(* IEC 61131-3 sources: beeguard/reference, 3 files *)

(* ---- analog_alarm.st ---- *)
FUNCTION_BLOCK BG_ALM_ANA
(*==========================================================================
BG_ALM_ANA - beeguard analog alarm.
Watches one REAL for up to six alarm conditions. Each condition is handled by
its own BG_ALM_DIG instance, so each one has the complete ISA-18.2 behaviour
(acknowledge, latch, shelve, priority, time stamps, count, chatter) and can be
acknowledged or shelved separately. Names follow BG_ALM_DIG (IN_, CFG_, CMD_OP_,
CMD_PG_, STS_, VAL_, TS_).

CONDITIONS (each enabled separately; HH and H may be in alarm at the same time)
	HH      above CFG_HH_SP; normal again below CFG_HH_SP - CFG_DEADBAND
	H       above CFG_H_SP;  normal again below CFG_H_SP  - CFG_DEADBAND
	L       below CFG_L_SP;  normal again above CFG_L_SP  + CFG_DEADBAND
	LL      below CFG_LL_SP; normal again above CFG_LL_SP + CFG_DEADBAND
	ROC_UP  rising faster than CFG_ROC_UP_SP units per second
	ROC_DN  falling faster than CFG_ROC_DN_SP units per second (enter it positive)
	The rate is measured once every CFG_ROC_PERIOD.

FILTERING
	Order: deadband, then on-delay, then off-delay (as recommended in
	ISA-TR18.2.3). The deadband and CFG_ON_DELAY_MS apply to the four limits;
	the rate conditions are filtered by CFG_ROC_PERIOD instead.
	CFG_OFF_DELAY_MS applies to all six. Typical starting points published in
	ISA-TR18.2.3 and EEMUA 191, to be tuned per loop: flow 5 % of span / 15 s,
	level 5 % / 60 s, pressure 2 % / 15 s, temperature 1 % / 60 s.

REQUESTS
	For one condition (one-shot): CMD_OP_<C>_ACK, CMD_OP_<C>_SHELVE,
	CMD_OP_<C>_UNSHELVE, where <C> is HH, H, L, LL, ROC_UP or ROC_DN.
	For all conditions (one-shot): CMD_OP_ACK_ALL, CMD_OP_RESET,
	CMD_OP_UNSHELVE_ALL, CMD_OP_DISABLE/ENABLE, CMD_OP_SUPPRESS/UNSUPPRESS.
	For all conditions from logic (rising edge): the CMD_PG_ equivalents.
	Suppression and out of service always cover the whole alarm. Read a
	condition's details from its instance, e.g. MYALARM.HH.TS_ALM.

VAL_DIAG bits
	.0 configuration fault (.2 to .5)      .3 CFG_DEADBAND is negative
	.1 IN_FAULT is set                     .4 rate settings invalid
	.2 enabled limits out of order         .5 a condition instance reports a fault
	   (must be LL <= L <= H <= HH)

BAD QUALITY
	While IN_FAULT is set the limit and rate checks keep their last result, and
	the rate measurement starts over once the value is good again.
==========================================================================*)
VAR_INPUT
	(* PROCESS *)
	IN_ENABLE: BOOL := TRUE;		// FALSE: THE BLOCK SKIPS ITS LOGIC AND OUTPUTS KEEP THEIR VALUES
	IN_VALUE: REAL;					// THE VALUE BEING ALARMED, IN ENGINEERING UNITS
	IN_FAULT: BOOL;					// IN_VALUE QUALITY IS BAD

	(* LIMITS *)
	CFG_HH_EN: BOOL;
	CFG_H_EN: BOOL;
	CFG_L_EN: BOOL;
	CFG_LL_EN: BOOL;
	CFG_HH_SP: REAL;
	CFG_H_SP: REAL;
	CFG_L_SP: REAL;
	CFG_LL_SP: REAL;
	CFG_DEADBAND: REAL;				// EU, APPLIED ON RETURN TO NORMAL

	(* RATE OF CHANGE *)
	CFG_ROC_UP_EN: BOOL;
	CFG_ROC_DN_EN: BOOL;
	CFG_ROC_UP_SP: REAL;			// EU/S RISE
	CFG_ROC_DN_SP: REAL;			// EU/S FALL, ENTERED AS A POSITIVE NUMBER
	CFG_ROC_PERIOD: TIME := T#1S;	// SAMPLE INTERVAL FOR THE RATE

	(* SEVERITY 1..1000 PER CONDITION *)
	CFG_HH_SEVERITY: DINT := 750;
	CFG_H_SEVERITY: DINT := 500;
	CFG_L_SEVERITY: DINT := 500;
	CFG_LL_SEVERITY: DINT := 750;
	CFG_ROC_UP_SEVERITY: DINT := 500;
	CFG_ROC_DN_SEVERITY: DINT := 500;

	(* ALARM BEHAVIOUR - SHARED BY ALL CONDITIONS *)
	CFG_ACK_REQ: BOOL := TRUE;
	CFG_LATCH: BOOL;
	CFG_ON_DELAY_MS: DINT;		// ON-DELAY (ms) FOR HH/H/L/LL
	CFG_OFF_DELAY_MS: DINT;			// OFF-DELAY (ms) FOR ALL CONDITIONS
	CFG_SHELVE_MAX: TIME;	// T#0S = SHELVING NOT PERMITTED
	CMD_SHELVE_TIME: TIME;		// T#0S = CFG_SHELVE_MAX
	CMD_SHELVE_ONESHOT: BOOL;
	CFG_CHATTER_COUNT: DINT;			// 0 = OFF
	CFG_CHATTER_WINDOW: TIME := T#60S;

	(* TIME STAMPING *)
	IN_CLOCK: DT;
	CFG_USE_SRC_TIME: BOOL;
	IN_SRC_TIME: DT;

	(* OPERATOR REQUESTS FOR ONE CONDITION - ONE-SHOT, CLEARED BY THE BLOCK *)
	CMD_OP_HH_ACK: BOOL;
	CMD_OP_H_ACK: BOOL;
	CMD_OP_L_ACK: BOOL;
	CMD_OP_LL_ACK: BOOL;
	CMD_OP_ROC_UP_ACK: BOOL;
	CMD_OP_ROC_DN_ACK: BOOL;
	CMD_OP_HH_SHELVE: BOOL;
	CMD_OP_H_SHELVE: BOOL;
	CMD_OP_L_SHELVE: BOOL;
	CMD_OP_LL_SHELVE: BOOL;
	CMD_OP_ROC_UP_SHELVE: BOOL;
	CMD_OP_ROC_DN_SHELVE: BOOL;
	CMD_OP_HH_UNSHELVE: BOOL;
	CMD_OP_H_UNSHELVE: BOOL;
	CMD_OP_L_UNSHELVE: BOOL;
	CMD_OP_LL_UNSHELVE: BOOL;
	CMD_OP_ROC_UP_UNSHELVE: BOOL;
	CMD_OP_ROC_DN_UNSHELVE: BOOL;

	(* OPERATOR REQUESTS FOR ALL CONDITIONS - ONE-SHOT, CLEARED BY THE BLOCK *)
	CMD_OP_ACK_ALL: BOOL;
	CMD_OP_RESET: BOOL;
	CMD_OP_UNSHELVE_ALL: BOOL;
	CMD_OP_DISABLE: BOOL;
	CMD_OP_ENABLE: BOOL;
	CMD_OP_SUPPRESS: BOOL;
	CMD_OP_UNSUPPRESS: BOOL;

	(* LOGIC REQUESTS FOR ALL CONDITIONS - RISING EDGE *)
	CMD_PG_ACK_ALL: BOOL;
	CMD_PG_RESET: BOOL;
	CMD_PG_UNSHELVE_ALL: BOOL;
	CMD_PG_DISABLE: BOOL;
	CMD_PG_ENABLE: BOOL;
	CMD_PG_SUPPRESS: BOOL;
	CMD_PG_UNSUPPRESS: BOOL;

	CMD_COUNT_RESET: BOOL;		// RISING EDGE, RESETS EVERY CONDITION'S COUNT
END_VAR
VAR_OUTPUT
	STS_ENABLED: BOOL;
	STS_ALM: BOOL;					// SOME CONDITION IS IN ALARM OR LATCHED
	STS_UNACKED: BOOL;				// SOME CONDITION WAITS FOR AN ACKNOWLEDGEMENT (HORN)
	STS_ALM_UNACK: BOOL;
	STS_ANY_SHELVED: BOOL;
	STS_SUPPRESSED: BOOL;
	STS_DISABLED: BOOL;
	STS_CHATTER: BOOL;				// SOME CONDITION IS CHATTERING
	STS_IN_FAULT: BOOL;
	STS_CFG_FAULT: BOOL;
	VAL_ACTIVE_PRIORITY: DINT;		// MOST URGENT PRIORITY CURRENTLY IN ALARM, 1..4. 0 = NONE
	VAL_ROC: REAL;					// LAST MEASURED RATE, UNITS PER SECOND
	VAL_DIAG: DINT;

	(* ONE INSTANCE PER CONDITION - READ THEIR OUTPUTS, DO NOT WRITE *)
	HH: BG_ALM_DIG;
	H: BG_ALM_DIG;
	L: BG_ALM_DIG;
	LL: BG_ALM_DIG;
	ROC_UP: BG_ALM_DIG;
	ROC_DN: BG_ALM_DIG;

	CFG_VERSION: REAL;
END_VAR
VAR
	HHCOND: BOOL;
	HCOND: BOOL;
	LCOND: BOOL;
	LLCOND: BOOL;
	ROCUPCOND: BOOL;
	ROCDNCOND: BOOL;

	ROC_TMR: TON;
	ROCLAST: REAL;
	ROCPRIMED: BOOL;			// ROCLAST HOLDS A GOOD SAMPLE

	LIMITPREV: REAL;
	LIMITSEEN: BOOL;
END_VAR

(*==========================================================================
Sets the Version of the Control Module on the HMI and in the Program.
==========================================================================
Date Last Updated: 10-1-2026
===========================================================================*)
//CFG_VERSION := 1.0; // ORIGINAL - ISA-18.2 ANALOG ALARM BUILT ON THE DIGITAL ALARM 3.0
CFG_VERSION := 1.1; //RENAMED BG_ALM_ANA WITH IN_/CFG_/CMD_/STS_/VAL_/TS_ NAMES; NO LOGIC CHANGE

STS_ENABLED := IN_ENABLE;
IF NOT IN_ENABLE THEN
	JMP CLEAR_COMMANDS;
END_IF

(*===========================================================================
CONFIGURATION - Enabled limits must be in order LL <= L <= H <= HH
===========================================================================*)
VAL_DIAG := 0;
LIMITSEEN := FALSE;
IF CFG_LL_EN THEN
	LIMITPREV := CFG_LL_SP;
	LIMITSEEN := TRUE;
END_IF
IF CFG_L_EN THEN
	IF LIMITSEEN AND CFG_L_SP < LIMITPREV THEN
		VAL_DIAG.2 := TRUE;
	END_IF
	LIMITPREV := CFG_L_SP;
	LIMITSEEN := TRUE;
END_IF
IF CFG_H_EN THEN
	IF LIMITSEEN AND CFG_H_SP < LIMITPREV THEN
		VAL_DIAG.2 := TRUE;
	END_IF
	LIMITPREV := CFG_H_SP;
	LIMITSEEN := TRUE;
END_IF
IF CFG_HH_EN THEN
	IF LIMITSEEN AND CFG_HH_SP < LIMITPREV THEN
		VAL_DIAG.2 := TRUE;
	END_IF
END_IF

VAL_DIAG.3 := CFG_DEADBAND < 0.0;
VAL_DIAG.4 := (CFG_ROC_UP_EN OR CFG_ROC_DN_EN) AND
	(CFG_ROC_PERIOD = T#0S OR CFG_ROC_UP_SP < 0.0 OR CFG_ROC_DN_SP < 0.0);

(*===========================================================================
LIMIT CONDITIONS - Deadband on return to normal. Held while IN_FAULT.
===========================================================================*)
STS_IN_FAULT := IN_FAULT;
IF NOT IN_FAULT THEN
	IF IN_VALUE > CFG_HH_SP THEN
		HHCOND := TRUE;
	ELSIF IN_VALUE < CFG_HH_SP - CFG_DEADBAND THEN
		HHCOND := FALSE;
	END_IF

	IF IN_VALUE > CFG_H_SP THEN
		HCOND := TRUE;
	ELSIF IN_VALUE < CFG_H_SP - CFG_DEADBAND THEN
		HCOND := FALSE;
	END_IF

	IF IN_VALUE < CFG_L_SP THEN
		LCOND := TRUE;
	ELSIF IN_VALUE > CFG_L_SP + CFG_DEADBAND THEN
		LCOND := FALSE;
	END_IF

	IF IN_VALUE < CFG_LL_SP THEN
		LLCOND := TRUE;
	ELSIF IN_VALUE > CFG_LL_SP + CFG_DEADBAND THEN
		LLCOND := FALSE;
	END_IF
END_IF

(*===========================================================================
RATE OF CHANGE - Sampled every CFG_ROC_PERIOD. A fault restarts the sampling so
the jump between bad and good data is never measured as a rate.
===========================================================================*)
IF (CFG_ROC_UP_EN OR CFG_ROC_DN_EN) AND CFG_ROC_PERIOD > T#0S AND NOT IN_FAULT THEN
	ROC_TMR(IN := NOT ROC_TMR.Q, PT := CFG_ROC_PERIOD);
	IF NOT ROCPRIMED THEN
		ROCLAST := IN_VALUE;
		ROCPRIMED := TRUE;
	ELSIF ROC_TMR.Q THEN
		VAL_ROC := (IN_VALUE - ROCLAST) / (TIME_TO_REAL(CFG_ROC_PERIOD) / 1000.0);
		ROCLAST := IN_VALUE;
		ROCUPCOND := VAL_ROC > CFG_ROC_UP_SP;
		ROCDNCOND := VAL_ROC < -CFG_ROC_DN_SP;
	END_IF
ELSE
	ROC_TMR(IN := FALSE);
	ROCPRIMED := FALSE;
	IF NOT IN_FAULT THEN
		VAL_ROC := 0.0;
		ROCUPCOND := FALSE;
		ROCDNCOND := FALSE;
	END_IF
END_IF

(*===========================================================================
CONDITION ALARMS - One BG_ALM_DIG per condition
===========================================================================*)
HH(IN_SIGNAL := CFG_HH_EN AND HHCOND, IN_FAULT := IN_FAULT, CFG_SEVERITY := CFG_HH_SEVERITY,
	CFG_ACK_REQ := CFG_ACK_REQ, CFG_LATCH := CFG_LATCH, CFG_ON_DELAY_MS := CFG_ON_DELAY_MS, CFG_OFF_DELAY_MS := CFG_OFF_DELAY_MS,
	CFG_SHELVE_MAX := CFG_SHELVE_MAX, CMD_SHELVE_TIME := CMD_SHELVE_TIME, CMD_SHELVE_ONESHOT := CMD_SHELVE_ONESHOT,
	CFG_CHATTER_COUNT := CFG_CHATTER_COUNT, CFG_CHATTER_WINDOW := CFG_CHATTER_WINDOW,
	IN_CLOCK := IN_CLOCK, CFG_USE_SRC_TIME := CFG_USE_SRC_TIME, IN_SRC_TIME := IN_SRC_TIME,
	CMD_OP_ACK := CMD_OP_HH_ACK OR CMD_OP_ACK_ALL, CMD_OP_RESET := CMD_OP_RESET,
	CMD_OP_SHELVE := CMD_OP_HH_SHELVE, CMD_OP_UNSHELVE := CMD_OP_HH_UNSHELVE OR CMD_OP_UNSHELVE_ALL,
	CMD_OP_DISABLE := CMD_OP_DISABLE, CMD_OP_ENABLE := CMD_OP_ENABLE, CMD_OP_SUPPRESS := CMD_OP_SUPPRESS, CMD_OP_UNSUPPRESS := CMD_OP_UNSUPPRESS,
	CMD_PG_ACK := CMD_PG_ACK_ALL, CMD_PG_RESET := CMD_PG_RESET, CMD_PG_UNSHELVE := CMD_PG_UNSHELVE_ALL,
	CMD_PG_DISABLE := CMD_PG_DISABLE, CMD_PG_ENABLE := CMD_PG_ENABLE, CMD_PG_SUPPRESS := CMD_PG_SUPPRESS, CMD_PG_UNSUPPRESS := CMD_PG_UNSUPPRESS,
	CMD_COUNT_RESET := CMD_COUNT_RESET);

H(IN_SIGNAL := CFG_H_EN AND HCOND, IN_FAULT := IN_FAULT, CFG_SEVERITY := CFG_H_SEVERITY,
	CFG_ACK_REQ := CFG_ACK_REQ, CFG_LATCH := CFG_LATCH, CFG_ON_DELAY_MS := CFG_ON_DELAY_MS, CFG_OFF_DELAY_MS := CFG_OFF_DELAY_MS,
	CFG_SHELVE_MAX := CFG_SHELVE_MAX, CMD_SHELVE_TIME := CMD_SHELVE_TIME, CMD_SHELVE_ONESHOT := CMD_SHELVE_ONESHOT,
	CFG_CHATTER_COUNT := CFG_CHATTER_COUNT, CFG_CHATTER_WINDOW := CFG_CHATTER_WINDOW,
	IN_CLOCK := IN_CLOCK, CFG_USE_SRC_TIME := CFG_USE_SRC_TIME, IN_SRC_TIME := IN_SRC_TIME,
	CMD_OP_ACK := CMD_OP_H_ACK OR CMD_OP_ACK_ALL, CMD_OP_RESET := CMD_OP_RESET,
	CMD_OP_SHELVE := CMD_OP_H_SHELVE, CMD_OP_UNSHELVE := CMD_OP_H_UNSHELVE OR CMD_OP_UNSHELVE_ALL,
	CMD_OP_DISABLE := CMD_OP_DISABLE, CMD_OP_ENABLE := CMD_OP_ENABLE, CMD_OP_SUPPRESS := CMD_OP_SUPPRESS, CMD_OP_UNSUPPRESS := CMD_OP_UNSUPPRESS,
	CMD_PG_ACK := CMD_PG_ACK_ALL, CMD_PG_RESET := CMD_PG_RESET, CMD_PG_UNSHELVE := CMD_PG_UNSHELVE_ALL,
	CMD_PG_DISABLE := CMD_PG_DISABLE, CMD_PG_ENABLE := CMD_PG_ENABLE, CMD_PG_SUPPRESS := CMD_PG_SUPPRESS, CMD_PG_UNSUPPRESS := CMD_PG_UNSUPPRESS,
	CMD_COUNT_RESET := CMD_COUNT_RESET);

L(IN_SIGNAL := CFG_L_EN AND LCOND, IN_FAULT := IN_FAULT, CFG_SEVERITY := CFG_L_SEVERITY,
	CFG_ACK_REQ := CFG_ACK_REQ, CFG_LATCH := CFG_LATCH, CFG_ON_DELAY_MS := CFG_ON_DELAY_MS, CFG_OFF_DELAY_MS := CFG_OFF_DELAY_MS,
	CFG_SHELVE_MAX := CFG_SHELVE_MAX, CMD_SHELVE_TIME := CMD_SHELVE_TIME, CMD_SHELVE_ONESHOT := CMD_SHELVE_ONESHOT,
	CFG_CHATTER_COUNT := CFG_CHATTER_COUNT, CFG_CHATTER_WINDOW := CFG_CHATTER_WINDOW,
	IN_CLOCK := IN_CLOCK, CFG_USE_SRC_TIME := CFG_USE_SRC_TIME, IN_SRC_TIME := IN_SRC_TIME,
	CMD_OP_ACK := CMD_OP_L_ACK OR CMD_OP_ACK_ALL, CMD_OP_RESET := CMD_OP_RESET,
	CMD_OP_SHELVE := CMD_OP_L_SHELVE, CMD_OP_UNSHELVE := CMD_OP_L_UNSHELVE OR CMD_OP_UNSHELVE_ALL,
	CMD_OP_DISABLE := CMD_OP_DISABLE, CMD_OP_ENABLE := CMD_OP_ENABLE, CMD_OP_SUPPRESS := CMD_OP_SUPPRESS, CMD_OP_UNSUPPRESS := CMD_OP_UNSUPPRESS,
	CMD_PG_ACK := CMD_PG_ACK_ALL, CMD_PG_RESET := CMD_PG_RESET, CMD_PG_UNSHELVE := CMD_PG_UNSHELVE_ALL,
	CMD_PG_DISABLE := CMD_PG_DISABLE, CMD_PG_ENABLE := CMD_PG_ENABLE, CMD_PG_SUPPRESS := CMD_PG_SUPPRESS, CMD_PG_UNSUPPRESS := CMD_PG_UNSUPPRESS,
	CMD_COUNT_RESET := CMD_COUNT_RESET);

LL(IN_SIGNAL := CFG_LL_EN AND LLCOND, IN_FAULT := IN_FAULT, CFG_SEVERITY := CFG_LL_SEVERITY,
	CFG_ACK_REQ := CFG_ACK_REQ, CFG_LATCH := CFG_LATCH, CFG_ON_DELAY_MS := CFG_ON_DELAY_MS, CFG_OFF_DELAY_MS := CFG_OFF_DELAY_MS,
	CFG_SHELVE_MAX := CFG_SHELVE_MAX, CMD_SHELVE_TIME := CMD_SHELVE_TIME, CMD_SHELVE_ONESHOT := CMD_SHELVE_ONESHOT,
	CFG_CHATTER_COUNT := CFG_CHATTER_COUNT, CFG_CHATTER_WINDOW := CFG_CHATTER_WINDOW,
	IN_CLOCK := IN_CLOCK, CFG_USE_SRC_TIME := CFG_USE_SRC_TIME, IN_SRC_TIME := IN_SRC_TIME,
	CMD_OP_ACK := CMD_OP_LL_ACK OR CMD_OP_ACK_ALL, CMD_OP_RESET := CMD_OP_RESET,
	CMD_OP_SHELVE := CMD_OP_LL_SHELVE, CMD_OP_UNSHELVE := CMD_OP_LL_UNSHELVE OR CMD_OP_UNSHELVE_ALL,
	CMD_OP_DISABLE := CMD_OP_DISABLE, CMD_OP_ENABLE := CMD_OP_ENABLE, CMD_OP_SUPPRESS := CMD_OP_SUPPRESS, CMD_OP_UNSUPPRESS := CMD_OP_UNSUPPRESS,
	CMD_PG_ACK := CMD_PG_ACK_ALL, CMD_PG_RESET := CMD_PG_RESET, CMD_PG_UNSHELVE := CMD_PG_UNSHELVE_ALL,
	CMD_PG_DISABLE := CMD_PG_DISABLE, CMD_PG_ENABLE := CMD_PG_ENABLE, CMD_PG_SUPPRESS := CMD_PG_SUPPRESS, CMD_PG_UNSUPPRESS := CMD_PG_UNSUPPRESS,
	CMD_COUNT_RESET := CMD_COUNT_RESET);

// ROC CONDITIONS ARE ALREADY FILTERED BY CFG_ROC_PERIOD, SO THEY HAVE NO ON-DELAY.
ROC_UP(IN_SIGNAL := CFG_ROC_UP_EN AND ROCUPCOND, IN_FAULT := IN_FAULT, CFG_SEVERITY := CFG_ROC_UP_SEVERITY,
	CFG_ACK_REQ := CFG_ACK_REQ, CFG_LATCH := CFG_LATCH, CFG_ON_DELAY_MS := 0, CFG_OFF_DELAY_MS := CFG_OFF_DELAY_MS,
	CFG_SHELVE_MAX := CFG_SHELVE_MAX, CMD_SHELVE_TIME := CMD_SHELVE_TIME, CMD_SHELVE_ONESHOT := CMD_SHELVE_ONESHOT,
	CFG_CHATTER_COUNT := CFG_CHATTER_COUNT, CFG_CHATTER_WINDOW := CFG_CHATTER_WINDOW,
	IN_CLOCK := IN_CLOCK, CFG_USE_SRC_TIME := CFG_USE_SRC_TIME, IN_SRC_TIME := IN_SRC_TIME,
	CMD_OP_ACK := CMD_OP_ROC_UP_ACK OR CMD_OP_ACK_ALL, CMD_OP_RESET := CMD_OP_RESET,
	CMD_OP_SHELVE := CMD_OP_ROC_UP_SHELVE, CMD_OP_UNSHELVE := CMD_OP_ROC_UP_UNSHELVE OR CMD_OP_UNSHELVE_ALL,
	CMD_OP_DISABLE := CMD_OP_DISABLE, CMD_OP_ENABLE := CMD_OP_ENABLE, CMD_OP_SUPPRESS := CMD_OP_SUPPRESS, CMD_OP_UNSUPPRESS := CMD_OP_UNSUPPRESS,
	CMD_PG_ACK := CMD_PG_ACK_ALL, CMD_PG_RESET := CMD_PG_RESET, CMD_PG_UNSHELVE := CMD_PG_UNSHELVE_ALL,
	CMD_PG_DISABLE := CMD_PG_DISABLE, CMD_PG_ENABLE := CMD_PG_ENABLE, CMD_PG_SUPPRESS := CMD_PG_SUPPRESS, CMD_PG_UNSUPPRESS := CMD_PG_UNSUPPRESS,
	CMD_COUNT_RESET := CMD_COUNT_RESET);

ROC_DN(IN_SIGNAL := CFG_ROC_DN_EN AND ROCDNCOND, IN_FAULT := IN_FAULT, CFG_SEVERITY := CFG_ROC_DN_SEVERITY,
	CFG_ACK_REQ := CFG_ACK_REQ, CFG_LATCH := CFG_LATCH, CFG_ON_DELAY_MS := 0, CFG_OFF_DELAY_MS := CFG_OFF_DELAY_MS,
	CFG_SHELVE_MAX := CFG_SHELVE_MAX, CMD_SHELVE_TIME := CMD_SHELVE_TIME, CMD_SHELVE_ONESHOT := CMD_SHELVE_ONESHOT,
	CFG_CHATTER_COUNT := CFG_CHATTER_COUNT, CFG_CHATTER_WINDOW := CFG_CHATTER_WINDOW,
	IN_CLOCK := IN_CLOCK, CFG_USE_SRC_TIME := CFG_USE_SRC_TIME, IN_SRC_TIME := IN_SRC_TIME,
	CMD_OP_ACK := CMD_OP_ROC_DN_ACK OR CMD_OP_ACK_ALL, CMD_OP_RESET := CMD_OP_RESET,
	CMD_OP_SHELVE := CMD_OP_ROC_DN_SHELVE, CMD_OP_UNSHELVE := CMD_OP_ROC_DN_UNSHELVE OR CMD_OP_UNSHELVE_ALL,
	CMD_OP_DISABLE := CMD_OP_DISABLE, CMD_OP_ENABLE := CMD_OP_ENABLE, CMD_OP_SUPPRESS := CMD_OP_SUPPRESS, CMD_OP_UNSUPPRESS := CMD_OP_UNSUPPRESS,
	CMD_PG_ACK := CMD_PG_ACK_ALL, CMD_PG_RESET := CMD_PG_RESET, CMD_PG_UNSHELVE := CMD_PG_UNSHELVE_ALL,
	CMD_PG_DISABLE := CMD_PG_DISABLE, CMD_PG_ENABLE := CMD_PG_ENABLE, CMD_PG_SUPPRESS := CMD_PG_SUPPRESS, CMD_PG_UNSUPPRESS := CMD_PG_UNSUPPRESS,
	CMD_COUNT_RESET := CMD_COUNT_RESET);

(*===========================================================================
OUTPUT UPDATES - Summary of all conditions
===========================================================================*)
STS_ALM := HH.STS_ALM OR H.STS_ALM OR L.STS_ALM OR LL.STS_ALM OR ROC_UP.STS_ALM OR ROC_DN.STS_ALM;
STS_UNACKED := HH.STS_UNACKED OR H.STS_UNACKED OR L.STS_UNACKED OR LL.STS_UNACKED OR ROC_UP.STS_UNACKED OR ROC_DN.STS_UNACKED;
STS_ALM_UNACK := HH.STS_ALM_UNACK OR H.STS_ALM_UNACK OR L.STS_ALM_UNACK OR LL.STS_ALM_UNACK
	OR ROC_UP.STS_ALM_UNACK OR ROC_DN.STS_ALM_UNACK;
STS_ANY_SHELVED := HH.STS_SHELVED OR H.STS_SHELVED OR L.STS_SHELVED OR LL.STS_SHELVED OR ROC_UP.STS_SHELVED OR ROC_DN.STS_SHELVED;
STS_CHATTER := HH.STS_CHATTER OR H.STS_CHATTER OR L.STS_CHATTER OR LL.STS_CHATTER
	OR ROC_UP.STS_CHATTER OR ROC_DN.STS_CHATTER;
STS_SUPPRESSED := HH.STS_SUPPRESSED;	// SUPPRESSION AND OUT OF SERVICE ARE SENT TO EVERY CONDITION
STS_DISABLED := HH.STS_DISABLED;

VAL_ACTIVE_PRIORITY := 0;
IF HH.STS_ALM AND (VAL_ACTIVE_PRIORITY = 0 OR HH.VAL_PRIORITY < VAL_ACTIVE_PRIORITY) THEN
	VAL_ACTIVE_PRIORITY := HH.VAL_PRIORITY;
END_IF
IF H.STS_ALM AND (VAL_ACTIVE_PRIORITY = 0 OR H.VAL_PRIORITY < VAL_ACTIVE_PRIORITY) THEN
	VAL_ACTIVE_PRIORITY := H.VAL_PRIORITY;
END_IF
IF L.STS_ALM AND (VAL_ACTIVE_PRIORITY = 0 OR L.VAL_PRIORITY < VAL_ACTIVE_PRIORITY) THEN
	VAL_ACTIVE_PRIORITY := L.VAL_PRIORITY;
END_IF
IF LL.STS_ALM AND (VAL_ACTIVE_PRIORITY = 0 OR LL.VAL_PRIORITY < VAL_ACTIVE_PRIORITY) THEN
	VAL_ACTIVE_PRIORITY := LL.VAL_PRIORITY;
END_IF
IF ROC_UP.STS_ALM AND (VAL_ACTIVE_PRIORITY = 0 OR ROC_UP.VAL_PRIORITY < VAL_ACTIVE_PRIORITY) THEN
	VAL_ACTIVE_PRIORITY := ROC_UP.VAL_PRIORITY;
END_IF
IF ROC_DN.STS_ALM AND (VAL_ACTIVE_PRIORITY = 0 OR ROC_DN.VAL_PRIORITY < VAL_ACTIVE_PRIORITY) THEN
	VAL_ACTIVE_PRIORITY := ROC_DN.VAL_PRIORITY;
END_IF

VAL_DIAG.1 := IN_FAULT;
VAL_DIAG.5 := HH.STS_CFG_FAULT OR H.STS_CFG_FAULT OR L.STS_CFG_FAULT OR LL.STS_CFG_FAULT
	OR ROC_UP.STS_CFG_FAULT OR ROC_DN.STS_CFG_FAULT;
STS_CFG_FAULT := VAL_DIAG.2 OR VAL_DIAG.3 OR VAL_DIAG.4 OR VAL_DIAG.5;
VAL_DIAG.0 := STS_CFG_FAULT;

(*===========================================================================
CLEAR OPERATOR REQUESTS - They are one-shot
===========================================================================*)
CLEAR_COMMANDS:
CMD_OP_HH_ACK := FALSE;
CMD_OP_H_ACK := FALSE;
CMD_OP_L_ACK := FALSE;
CMD_OP_LL_ACK := FALSE;
CMD_OP_ROC_UP_ACK := FALSE;
CMD_OP_ROC_DN_ACK := FALSE;
CMD_OP_HH_SHELVE := FALSE;
CMD_OP_H_SHELVE := FALSE;
CMD_OP_L_SHELVE := FALSE;
CMD_OP_LL_SHELVE := FALSE;
CMD_OP_ROC_UP_SHELVE := FALSE;
CMD_OP_ROC_DN_SHELVE := FALSE;
CMD_OP_HH_UNSHELVE := FALSE;
CMD_OP_H_UNSHELVE := FALSE;
CMD_OP_L_UNSHELVE := FALSE;
CMD_OP_LL_UNSHELVE := FALSE;
CMD_OP_ROC_UP_UNSHELVE := FALSE;
CMD_OP_ROC_DN_UNSHELVE := FALSE;
CMD_OP_ACK_ALL := FALSE;
CMD_OP_RESET := FALSE;
CMD_OP_UNSHELVE_ALL := FALSE;
CMD_OP_DISABLE := FALSE;
CMD_OP_ENABLE := FALSE;
CMD_OP_SUPPRESS := FALSE;
CMD_OP_UNSUPPRESS := FALSE;

END_FUNCTION_BLOCK

(* ---- analog_v2.1.st ---- *)
FUNCTION_BLOCK AOI_CM_AIN
VAR_INPUT
	IN_IOH: BOOL;
	IN_INH1: DINT;
	IN_OVR: BOOL;
	IN_UNR: BOOL;
	IN_RAW: REAL;
	CMD_ALM_RES: BOOL;
END_VAR
VAR_INPUT PERSISTENT RETAIN
	CFG_EN: BOOL;
	CFG_RU_MAX: DINT;
	CFG_RU_MIN: DINT;
	CFG_EU_MAX: REAL;
	CFG_EU_MIN: REAL;
	CFG_HIHI_SP: REAL;
	CFG_HI_SP: REAL;
	CFG_LO_SP: REAL;
	CFG_LOLO_SP: REAL;
	CFG_FRZN_SP: REAL;
	CFG_DEC_PT: DINT;
	CFG_DESC: STRING;
	CFG_DEV_TYPE: DINT;
	CFG_EID: STRING;
	CFG_EN_ALM_HI: BOOL;
	CFG_EN_ALM_HIHI: BOOL;
	CFG_EN_ALM_IOH: BOOL;
	CFG_EN_ALM_LO: BOOL;
	CFG_EN_ALM_LOLO: BOOL;
	CFG_EN_ALM_OOR: BOOL;
	CFG_EN_ALM_FRZN: BOOL;
	CFG_EN_IOH: BOOL;
	CFG_EN_OOR: BOOL;
	CFG_EN_SCL: BOOL;
	CFG_EN_TOT: BOOL;
	CFG_EN_FRZN: BOOL;
	CFG_HI_DT: DINT;
	CFG_HIHI_DT: DINT;
	CFG_LO_DT: DINT;
	CFG_LOLO_DT: DINT;
	CFG_OOR_DT: DINT;
	CFG_FRZN_DT: DINT;
	CFG_SCL_TYP: DINT;
	CFG_UNITS: STRING;
	SIM: BOOL;
	CFG_TMR_DISABLE_SIM: BOOL;
END_VAR
VAR_IN_OUT
	ALMD_HIHI: AOI_CM_ALMD;
	ALMD_HI: AOI_CM_ALMD;
	ALMD_LO: AOI_CM_ALMD;
	ALMD_LOLO: AOI_CM_ALMD;
	ALMD_OOR: AOI_CM_ALMD;
	ALMD_IOH: AOI_CM_ALMD;
	ALMD_FRZN: AOI_CM_ALMD;
END_VAR
VAR_OUTPUT
	STS_RDY2GO: BOOL;
	VAL_ACT: REAL;
	ALM_HIHI: BOOL;
	ALM_HI: BOOL;
	ALM_LO: BOOL;
	ALM_LOLO: BOOL;
	ALM_OOR: BOOL;
	ALM_IOH: BOOL;
	ALM_FRZN: BOOL;
	STS_HIHI: BOOL;
	STS_HI: BOOL;
	STS_LO: BOOL;
	STS_LOLO: BOOL;
	STS_OOR: BOOL;
	STS_IOH: BOOL;
	STS_FRZN: BOOL;
	CFG_VERSION: REAL;
	STS_ALM_ANY: BOOL;
	STS_ALM_ANY_UNACK: BOOL;
	ALM_ANY: BOOL;
	VAL_S: DINT;
END_VAR
VAR
	SIM_ONS: R_TRIG;
	WRK_B0: BOOL;
	WRK_B1: BOOL;
	WRK_ONS: ARRAY[0..15] OF R_TRIG;
	WRK_R: ARRAY[0..6] OF REAL;
	WRK_T: ARRAY[0..7] OF TON;
END_VAR

(*===========================================================================
AOI: CM_AIN
Date Last Updated: 5-27-2024
===========================================================================*)
//CFG_VERSION:= 1.0; // ORIGINAL
//CFG_VERSION := 2.0; //ADDED AOI_CM_ALMD FUNCTION BLOCK
CFG_VERSION := 2.1; //ADDED FRONZEN DATA ALARM LOGIC
(*===========================================================================
RETURN IF DISABLED  - If Module is Disabled, Scan One Last Time for Cleanup, Then Return
===========================================================================*)
IF NOT(CFG_EN) THEN
	WRK_ONS[1].CLK := TRUE;
	IF WRK_ONS[1].Q THEN
		WRK_B1 := TRUE;
	END_IF
	IF NOT(WRK_B1) THEN
		JMP EXIT_AOI_CM_AIN;
	END_IF
ELSE
	WRK_B1 := FALSE;
	WRK_ONS[1].CLK := FALSE;
END_IF

(*===========================================================================
SETUP - Clean up the Config: Enable Alarming depending on what Inputs are Confirmed in the System.
===========================================================================*)
IF NOT(CFG_EN_IOH) THEN
	CFG_EN_ALM_IOH := FALSE;
END_IF
IF NOT(CFG_EN_OOR) THEN
	CFG_EN_ALM_OOR := FALSE;
END_IF
IF NOT(CFG_EN_FRZN) THEN
	CFG_EN_ALM_FRZN := FALSE;
END_IF
(*===========================================================================
SETUP - Prevent wire-framing in HMI during start up (this prevents dividing by zero).
===========================================================================*)
IF CFG_EU_MAX = 0.0 THEN
	CFG_EU_MAX := 100;
END_IF

(*===========================================================================
TIMER PRESETS - Check and correct for invalid Timer Preset values
===========================================================================*)
WRK_T[1].PT := DINT_TO_TIME(ABS(CFG_HIHI_DT)*1000);
WRK_T[2].PT := DINT_TO_TIME(ABS(CFG_HI_DT)*1000);
WRK_T[3].PT := DINT_TO_TIME(ABS(CFG_LO_DT)*1000);
WRK_T[4].PT := DINT_TO_TIME(ABS(CFG_LOLO_DT)*1000);
WRK_T[5].PT := DINT_TO_TIME(ABS(CFG_OOR_DT)*1000);
WRK_T[7].PT := DINT_TO_TIME(ABS(CFG_FRZN_DT)*1000);

(*===========================================================================
COMMANDS - Latch Internal Work Bit To Clear All Alarms
===========================================================================*)
SIM_ONS.CLK := SIM;
IF CMD_ALM_RES OR (SIM_ONS.Q) THEN
	WRK_B0 := TRUE;
	CMD_ALM_RES := FALSE;
END_IF

(*===========================================================================
STATUS - I/O Health
===========================================================================*)
IF (CFG_EN_IOH AND IN_IOH) OR (NOT(CFG_EN_IOH)) OR (SIM) THEN
	STS_IOH := TRUE;
ELSE
	STS_IOH := FALSE;
END_IF

(*===========================================================================
STATUS - I/O Health
===========================================================================*)
IF (CFG_EN_OOR) AND (IN_OVR OR IN_UNR) THEN
	STS_OOR := TRUE;
ELSE
	STS_OOR := FALSE;
END_IF

(*===========================================================================
STATUS  - CM Ready to Go
CM is Ready to Go if it is Enabled, it's HOA(s) are in the Auto position and Interlocks are met.
NOTE: Not all conditions may exist for a given CM Cla
===========================================================================*)
IF (CFG_EN AND STS_IOH) THEN
	STS_RDY2GO := TRUE;
ELSE
	STS_RDY2GO := FALSE;
END_IF

(*===========================================================================
ALARMS HIHI - Determine HIHI Alarm if Alarms are Enabled.  If an Alarm is already
present when it is Disabled becomes it will stay TRUE.
===========================================================================*)
IF (VAL_ACT > CFG_HIHI_SP) THEN
	WRK_T[1](IN := TRUE);
	IF WRK_T[1].Q THEN
		STS_HIHI := TRUE;
		IF NOT(IN_INH1.0) AND CFG_EN_ALM_HIHI THEN
			ALM_HIHI := TRUE;
		ELSE
			ALM_HIHI := FALSE;
		END_IF
	ELSE
		STS_HIHI := FALSE;
	END_IF
ELSE
	STS_HIHI := FALSE;
	ALM_HIHI := FALSE;
	WRK_T[1](IN := FALSE);
END_IF

IF CFG_EN_ALM_HIHI AND ALM_HIHI AND NOT(IN_INH1.0) THEN
	ALMD_HIHI(IN := TRUE, ACKREQUIRED:=TRUE,LATCHED:=TRUE,MINDURATIONPRE:=1000);
ELSE
	ALMD_HIHI(IN := FALSE);
END_IF

IF WRK_B0 THEN
	 WRK_ONS[5].CLK := TRUE;
	 IF WRK_ONS[5].Q THEN
		 ALMD_HIHI.OPERACK := TRUE;
	 END_IF
ELSE
	WRK_ONS[5].CLK := FALSE;
END_IF

(*===========================================================================
ALARMS HI - Determine HI Alarm if Alarms are Enabled.  If an Alarm is already
present when it is Disabled becomes it will stay TRUE.
===========================================================================*)
IF (VAL_ACT > CFG_HI_SP) THEN
	WRK_T[2](IN := TRUE);
	IF WRK_T[2].Q THEN
		STS_HI := TRUE;
		IF NOT(IN_INH1.1) AND CFG_EN_ALM_HI THEN
			ALM_HI := TRUE;
		ELSE
			ALM_HI := FALSE;
		END_IF
	ELSE
		STS_HI := FALSE;
	END_IF
ELSE
	STS_HI := FALSE;
	ALM_HI := FALSE;
	WRK_T[2](IN := FALSE);
END_IF

IF CFG_EN_ALM_HI AND ALM_HI AND NOT(IN_INH1.1) THEN
	ALMD_HI(IN := TRUE, ACKREQUIRED:=TRUE,LATCHED:=TRUE,MINDURATIONPRE:=1000);
ELSE
	ALMD_HI(IN := FALSE);
END_IF

IF WRK_B0 THEN
	 WRK_ONS[7].CLK := TRUE;
	 IF WRK_ONS[7].Q THEN
		 ALMD_HI.OPERACK := TRUE;
	 END_IF
ELSE
	WRK_ONS[7].CLK := FALSE;
END_IF

(*===========================================================================
ALARMS LO - Determine LO Alarm if Alarms are Enabled.  If an Alarm is already
present when it is Disabled becomes it will stay TRUE.
===========================================================================*)
IF (VAL_ACT < CFG_LO_SP) THEN
	WRK_T[3](IN := TRUE);
	IF WRK_T[3].Q THEN
		STS_LO := TRUE;
		IF NOT(IN_INH1.2) AND CFG_EN_ALM_LO THEN
			ALM_LO := TRUE;
		ELSE
			ALM_LO := FALSE;
		END_IF
	ELSE
		STS_LO := FALSE;
	END_IF
ELSE
	STS_LO := FALSE;
	ALM_LO := FALSE;
	WRK_T[3](IN := FALSE);
END_IF

IF CFG_EN_ALM_LO AND ALM_LO AND NOT(IN_INH1.2) THEN
	ALMD_LO(IN := TRUE, ACKREQUIRED:=TRUE,LATCHED:=TRUE,MINDURATIONPRE:=1000);
ELSE
	ALMD_LO(IN := FALSE);
END_IF

IF WRK_B0 THEN
	 WRK_ONS[9].CLK := TRUE;
	 IF WRK_ONS[9].Q THEN
		 ALMD_LO.OPERACK := TRUE;
	 END_IF
ELSE
	WRK_ONS[9].CLK := FALSE;
END_IF

(*===========================================================================
ALARMS LOLO - Determine LOLO Alarm if Alarms are Enabled.  If an Alarm is already
present when it is Disabled becomes it will stay TRUE.
===========================================================================*)
IF (VAL_ACT < CFG_LOLO_SP) THEN
	WRK_T[4](IN := TRUE);
	IF WRK_T[4].Q THEN
		STS_LOLO := TRUE;
		IF NOT(IN_INH1.3) AND CFG_EN_ALM_LOLO THEN
			ALM_LOLO := TRUE;
		ELSE
			ALM_LOLO := FALSE;
		END_IF
	ELSE
		STS_LOLO := FALSE;
	END_IF
ELSE
	STS_LOLO := FALSE;
	ALM_LOLO := FALSE;
	WRK_T[4](IN := FALSE);
END_IF

IF CFG_EN_ALM_LOLO AND ALM_LOLO AND NOT(IN_INH1.3) THEN
	ALMD_LOLO(IN := TRUE, ACKREQUIRED:=TRUE,LATCHED:=TRUE,MINDURATIONPRE:=1000);
ELSE
	ALMD_LOLO(IN := FALSE);
END_IF

IF WRK_B0 THEN
	 WRK_ONS[11].CLK := TRUE;
	 IF WRK_ONS[11].Q THEN
		 ALMD_LOLO.OPERACK := TRUE;
	 END_IF
ELSE
	WRK_ONS[11].CLK := FALSE;
END_IF

(*===========================================================================
ALARMS - Out of Range
===========================================================================*)
IF (CFG_EN_ALM_OOR AND STS_OOR) THEN
	WRK_T[5](IN := TRUE);
	IF WRK_T[5].Q THEN
		//STS_OOR := TRUE; SEE LINE 35
		IF NOT(IN_INH1.4) THEN
			ALM_OOR := TRUE;
		ELSE
			ALM_OOR := FALSE;
		END_IF
	END_IF
ELSE
	ALM_OOR := FALSE;
	WRK_T[5](IN := FALSE);
END_IF

IF CFG_EN_ALM_OOR AND ALM_OOR AND NOT(IN_INH1.4) THEN
	ALMD_OOR(IN := TRUE, ACKREQUIRED:=TRUE,LATCHED:=TRUE,MINDURATIONPRE:=1000);
ELSE
	ALMD_OOR(IN := FALSE);
END_IF

IF WRK_B0 THEN
	 WRK_ONS[13].CLK := TRUE;
	 IF WRK_ONS[13].Q THEN
		 ALMD_OOR.OPERACK := TRUE;
	 END_IF
ELSE
	WRK_ONS[13].CLK := FALSE;
END_IF

(*===========================================================================
ALARMS - FROZEN VALUE
===========================================================================*)
IF (VAL_ACT = CFG_FRZN_SP) THEN
	STS_FRZN := TRUE;
ELSE
	STS_FRZN := FALSE;
END_IF

IF (CFG_EN_ALM_FRZN AND STS_FRZN) THEN
	WRK_T[7](IN := TRUE);
	IF WRK_T[7].Q THEN
		//STS_FRZN := TRUE; SEE LINE 35
		IF NOT(IN_INH1.5)THEN
			ALM_FRZN := TRUE;
		ELSE
			ALM_FRZN := FALSE;
		END_IF
	END_IF
ELSE
	ALM_FRZN := FALSE;
	WRK_T[7](IN := FALSE);
END_IF

IF WRK_T[7].ET > T#0S OR CFG_EN_ALM_FRZN THEN
	CFG_FRZN_SP := VAL_ACT;
END_IF

IF CFG_EN_ALM_FRZN AND ALM_FRZN AND NOT(IN_INH1.5) THEN
	ALMD_FRZN(IN := TRUE, ACKREQUIRED:=TRUE,LATCHED:=TRUE,MINDURATIONPRE:=60000);
ELSE
	ALMD_FRZN(IN := FALSE);
END_IF

IF WRK_B0 THEN
	 WRK_ONS[14].CLK := TRUE;
	 IF WRK_ONS[14].Q THEN
		 ALMD_FRZN.OPERACK := TRUE;
	 END_IF
ELSE
	WRK_ONS[14].CLK := FALSE;
END_IF

(*===========================================================================
ALARM - I/O Health (Includes Module Health, Channel Calibration Fault, or Channel Fault Alarms)
===========================================================================*)
IF CFG_EN_ALM_IOH AND NOT(STS_IOH) AND NOT(IN_INH1.5) THEN
	ALM_IOH := TRUE;
ELSE
	ALM_IOH := FALSE;
END_IF

IF CFG_EN_ALM_IOH AND ALM_IOH AND NOT(IN_INH1.5) THEN
	ALMD_IOH(IN := TRUE, ACKREQUIRED:=TRUE,LATCHED:=TRUE,MINDURATIONPRE:=1000);
ELSE
	ALMD_IOH(IN := FALSE);
END_IF

IF WRK_B0 THEN
	 WRK_ONS[15].CLK := TRUE;
	 IF WRK_ONS[15].Q THEN
		 ALMD_IOH.OPERACK := TRUE;
	 END_IF
ELSE
	WRK_ONS[15].CLK := FALSE;
END_IF

(*===========================================================================
ALARMS - Any Alarm
===========================================================================*)
IF ALM_HIHI OR ALM_HI OR ALM_LO OR ALM_LOLO OR ALM_OOR OR ALM_IOH OR ALM_FRZN THEN
	ALM_ANY := TRUE;
	STS_ALM_ANY := TRUE;
ELSE
	ALM_ANY := FALSE;
	STS_ALM_ANY := FALSE;
END_IF

(*===========================================================================
ALARMS - Check to see if there are any unacknowledged alarms.
===========================================================================*)
IF (ALM_HIHI AND NOT ALMD_HIHI.ACKED) OR (ALM_HI AND NOT ALMD_HI.ACKED) OR (ALM_LO AND NOT ALMD_LO.ACKED) OR (ALM_LOLO AND NOT ALMD_LOLO.ACKED) OR (ALM_OOR AND NOT ALMD_OOR.ACKED) OR (ALM_IOH AND NOT ALMD_IOH.ACKED) OR (ALM_FRZN AND NOT ALMD_FRZN.ACKED) THEN
	STS_ALM_ANY_UNACK := TRUE;
ELSE
	STS_ALM_ANY_UNACK := FALSE;
END_IF

(*===========================================================================
VALUES - State (HMI Color)
0 = Normal
1 = In Alarm
2 = Disabled
===========================================================================*)
IF NOT ALM_ANY THEN
	VAL_S := 0;
END_IF
IF ALM_ANY AND STS_ALM_ANY_UNACK THEN
	VAL_S := 1;
END_IF
IF ALM_ANY AND NOT STS_ALM_ANY_UNACK THEN
	VAL_S := 3;
END_IF

(*===========================================================================
VALUES - Actual Value
===========================================================================*)
IF CFG_EN_SCL THEN
	// SCALING CONFIGURATION
	IF CFG_SCL_TYP <> 1 AND CFG_SCL_TYP <> 2 THEN
		CFG_SCL_TYP := 1;
	END_IF
	IF CFG_RU_MAX = 0 AND CFG_RU_MIN = 0 THEN
		CFG_RU_MAX := 20;
		CFG_RU_MIN := 4;
	END_IF
	IF CFG_EU_MAX = 0 THEN
		CFG_EU_MAX := 1;
	END_IF
	IF CFG_RU_MAX = 0 THEN
		CFG_RU_MAX := 1;
	END_IF
	// LINEAR SCALING
	IF CFG_SCL_TYP = 1 THEN
		IF CFG_RU_MAX > CFG_RU_MIN THEN
			WRK_R[4] := (IN_RAW - DINT_TO_REAL(CFG_RU_MIN))/DINT_TO_REAL(CFG_RU_MAX - CFG_RU_MIN) * (CFG_EU_MAX-CFG_EU_MIN)+CFG_EU_MIN;
		END_IF
	END_IF
	// NON-LINEAR SCALING CONFIGURATION
	IF CFG_SCL_TYP = 2 THEN
		IF CFG_EU_MIN >= 0 THEN
			WRK_R[1] := LREAL_TO_REAL(EXPT(CFG_EU_MIN, 2));
		END_IF
		IF CFG_EU_MIN < 0 THEN
			WRK_R[1] := LREAL_TO_REAL(-1.0*EXPT(CFG_EU_MIN, 2));
		END_IF
		IF CFG_EU_MAX >= 0 THEN
			WRK_R[2] := LREAL_TO_REAL(EXPT(CFG_EU_MAX, 2));
		END_IF
		IF CFG_EU_MAX < 0 THEN
			WRK_R[2] := LREAL_TO_REAL(-1.0*EXPT(CFG_EU_MAX, 2));
		END_IF
		// NON-LINEAR SCALING
		IF CFG_RU_MAX > CFG_RU_MIN THEN
			WRK_R[3] := (IN_RAW - DINT_TO_REAL(CFG_RU_MIN))* (WRK_R[2] - WRK_R[1])/ DINT_TO_REAL(CFG_RU_MAX-CFG_RU_MIN)+ WRK_R[1];
		END_IF
		IF WRK_R[3] >= 0 THEN
			WRK_R[4] := SQRT(WRK_R[3]);
		END_IF
		IF WRK_R[3] < 0 THEN
			WRK_R[4] := -1.0 * SQRT(WRK_R[3]);
		END_IF
	END_IF
END_IF

IF NOT CFG_EN_SCL THEN
	WRK_R[4] := IN_RAW;
END_IF

VAL_ACT := WRK_R[4];

IF SIM THEN
	VAL_ACT := WRK_R[5];
END_IF

(*===========================================================================
SIM - Don't let the SIM bit stay on for more than 24 hours.
ADDED - TIMER BYPASS: NOTE SIM IS FOREVER!!!!
===========================================================================*)
IF SIM AND NOT CFG_TMR_DISABLE_SIM THEN
	WRK_T[6](IN := TRUE, PT := T#1440000MS);
	IF WRK_T[6].Q THEN
		SIM := FALSE;
	END_IF
ELSE
	WRK_T[6](IN := FALSE);
END_IF

(*===========================================================================
Unlatch Alarms Reset Bit
===========================================================================*)
IF WRK_B0 THEN
	WRK_B0 := FALSE;
END_IF

(*===========================================================================
CM DISABLED - Set Conditions Upon Entering Disabled State
===========================================================================*)
IF WRK_B1 THEN
	WRK_B0 := FALSE;
	VAL_S := 3;
	SIM := FALSE;
END_IF

(*===========================================================================
Exit AOI
===========================================================================*)
EXIT_AOI_CM_AIN:

END_FUNCTION_BLOCK

(* ---- digital_alarm.st ---- *)
FUNCTION_BLOCK BG_ALM_DIG
(*==========================================================================
BG_ALM_DIG - beeguard digital alarm.
Implements the alarm states of ISA-18.2 / IEC 62682 for one BOOL signal.

NAMING
	IN_   process inputs            CMD_OP_  operator requests (one-shot)
	CFG_  configuration             CMD_PG_  logic requests (rising edge)
	STS_  BOOL status outputs       VAL_     numeric outputs
	TS_   event time stamps (DT)

VAL_STATE
	0 NORMAL          ISA A  signal normal, nothing to acknowledge
	1 ACTIVE_UNACK    ISA B  in alarm, not yet acknowledged
	2 ACTIVE_ACK      ISA C  in alarm, acknowledged
	3 RTN_UNACK       ISA D  back to normal before anyone acknowledged it
	4 LATCHED_UNACK   ISA E  latched, back to normal, not yet acknowledged
	5 LATCHED_ACK     ISA E  latched, acknowledged, needs CMD_*_RESET
	6 SHELVED         ISA F  hidden by an operator for a limited time
	7 SUPPRESSED      ISA G  hidden by design
	8 OUT_OF_SERVICE  ISA H  removed from service, e.g. for maintenance

HIDING
	While shelved, suppressed or out of service the alarm is neither shown nor
	counted, and its state rests at NORMAL. When it is shown again with the
	signal still in alarm, it starts over as ACTIVE_UNACK, so nothing that
	happened while it was hidden can go unnoticed.

REQUESTS
	CMD_OP_* come from an HMI and are cleared by this block once handled.
	CMD_PG_* come from logic and are taken on their rising edge.
	There is no CMD_PG_SHELVE: only an operator may shelve (ISA-18.2).
	If a request and its opposite arrive together, ENABLE, UNSUPPRESS and
	UNSHELVE take effect.

VAL_DIAG bits
	.0 configuration fault (.2, .3 or .4)  .4 chatter settings invalid
	.1 IN_FAULT is set                     .5 last shelve request refused
	.2 CFG_SEVERITY not in 1..1000         .6 chattering
	.3 a negative delay

RESTART
	Nothing here is retained. After a cold restart a signal that is still in
	alarm is announced again as ACTIVE_UNACK, and any shelve is gone.
==========================================================================*)
VAR_INPUT
	(* PROCESS *)
	IN_ENABLE: BOOL := TRUE;		// FALSE: THE BLOCK SKIPS ITS LOGIC AND OUTPUTS KEEP THEIR VALUES
	IN_SIGNAL: BOOL;				// THE SIGNAL BEING ALARMED
	IN_FAULT: BOOL;					// SIGNAL QUALITY IS BAD: KEEP THE LAST GOOD ALARM CONDITION
	CFG_INVERT: BOOL;				// FALSE: ALARM WHILE IN_SIGNAL IS TRUE. TRUE: ALARM WHILE IT IS FALSE

	(* CONFIGURATION *)
	CFG_ACK_REQ: BOOL;				// TRUE: AN OPERATOR MUST ACKNOWLEDGE
	CFG_LATCH: BOOL;				// TRUE: STAYS IN ALARM AFTER RETURN TO NORMAL UNTIL RESET
	CFG_ON_DELAY_MS: DINT;			// THE SIGNAL MUST BE IN ALARM THIS LONG (ms) BEFORE IT IS ANNOUNCED
	CFG_OFF_DELAY_MS: DINT;			// ...AND NORMAL THIS LONG (ms) BEFORE IT RETURNS TO NORMAL
	CFG_SEVERITY: DINT := 500;		// 1..1000; VAL_PRIORITY IS DERIVED FROM IT
	CFG_SHELVE_MAX: TIME;			// UPPER LIMIT FOR ANY SHELVE. T#0S: SHELVING IS NOT ALLOWED
	CMD_SHELVE_TIME: TIME;			// LENGTH OF THE NEXT SHELVE. T#0S: USE CFG_SHELVE_MAX
	CMD_SHELVE_ONESHOT: BOOL;		// THE NEXT SHELVE ALSO ENDS WHEN THE SIGNAL RETURNS TO NORMAL
	CFG_CHATTER_COUNT: DINT;		// THIS MANY ACTIVATIONS IN ONE CFG_CHATTER_WINDOW = CHATTERING. 0: OFF
	CFG_CHATTER_WINDOW: TIME := T#60S;

	(* TIME STAMPING *)
	IN_CLOCK: DT;					// WALL-CLOCK DATE AND TIME OF THE CONTROLLER
	CFG_USE_SRC_TIME: BOOL;			// TRUE: STAMP EVENTS WITH IN_SRC_TIME INSTEAD OF IN_CLOCK
	IN_SRC_TIME: DT;				// E.G. THE TIME AN SOE INPUT MODULE SAW THE CHANGE

	(* OPERATOR REQUESTS - ONE-SHOT, CLEARED BY THE BLOCK *)
	CMD_OP_ACK: BOOL;
	CMD_OP_RESET: BOOL;
	CMD_OP_DISABLE: BOOL;
	CMD_OP_ENABLE: BOOL;
	CMD_OP_SUPPRESS: BOOL;
	CMD_OP_UNSUPPRESS: BOOL;
	CMD_OP_SHELVE: BOOL;
	CMD_OP_UNSHELVE: BOOL;

	(* LOGIC REQUESTS - RISING EDGE *)
	CMD_PG_ACK: BOOL;
	CMD_PG_RESET: BOOL;
	CMD_PG_DISABLE: BOOL;
	CMD_PG_ENABLE: BOOL;
	CMD_PG_SUPPRESS: BOOL;
	CMD_PG_UNSUPPRESS: BOOL;
	CMD_PG_UNSHELVE: BOOL;

	CMD_COUNT_RESET: BOOL;		// RISING EDGE
END_VAR
VAR_OUTPUT
	STS_ENABLED: BOOL;
	STS_ALM: BOOL;					// IN ALARM OR LATCHED (VAL_STATE 1, 2, 4, 5)
	STS_ACKED: BOOL;				// NOTHING WAITS FOR AN ACKNOWLEDGEMENT
	STS_ALM_UNACK: BOOL;			// STS_ALM AND NOT STS_ACKED
	STS_UNACKED: BOOL;				// SOMETHING WAITS FOR AN ACKNOWLEDGEMENT, RTN_UNACK INCLUDED (HORN)
	STS_COND: BOOL;					// FILTERED ALARM CONDITION, REPORTED EVEN WHILE HIDDEN
	STS_SUPPRESSED: BOOL;
	STS_SHELVED: BOOL;
	STS_DISABLED: BOOL;
	STS_CHATTER: BOOL;
	STS_IN_FAULT: BOOL;
	STS_CFG_FAULT: BOOL;
	VAL_PRIORITY: DINT;				// 1 URGENT, 2 HIGH, 3 MEDIUM, 4 LOW
	VAL_COUNT: DINT;
	VAL_STATE: DINT;
	VAL_DIAG: DINT;

	TS_ALM: DT;
	TS_ACK: DT;
	TS_RTN: DT;
	TS_RESET: DT;
	TS_COUNT_RESET: DT;
	TS_SHELVE: DT;
	TS_UNSHELVE: DT;
	TS_SHELVE_EXPIRY: DT;
	VAL_SHELVE_LEFT: TIME;

	VAL_ON_DELAY_MS: DINT;			// TIME (ms) THE ON-DELAY HAS RUN SO FAR
	CFG_VERSION: REAL;
END_VAR
VAR
	ALMSTATE: DINT;				// BASE STATE 0..5
	NOW: DT;
	RAWCOND: BOOL;
	LASTGOODCOND: BOOL;
	COND: BOOL;					// CONDITION AFTER ON/OFF DELAY
	SHELVEPT: TIME;
	SHELVEDONESHOT: BOOL;
	SHELVEREJECTED: BOOL;
	CHATTERACC: DINT;

	ACKCMD: BOOL;
	RESETCMD: BOOL;
	DISABLECMD: BOOL;
	ENABLECMD: BOOL;
	SUPPRESSCMD: BOOL;
	UNSUPPRESSCMD: BOOL;
	SHELVECMD: BOOL;
	UNSHELVECMD: BOOL;

	ON_TMR: TON;
	OFF_TMR: TON;
	SHELVE_TMR: TON;
	CHATTER_TMR: TON;
	COND_RISE: R_TRIG;
	COND_FALL: F_TRIG;
	PG_ACK_ONS: R_TRIG;
	PG_RESET_ONS: R_TRIG;
	PG_DISABLE_ONS: R_TRIG;
	PG_ENABLE_ONS: R_TRIG;
	PG_SUPPRESS_ONS: R_TRIG;
	PG_UNSUPPRESS_ONS: R_TRIG;
	PG_UNSHELVE_ONS: R_TRIG;
	COUNTRESET_ONS: R_TRIG;
END_VAR
VAR CONSTANT
	ST_NORMAL: DINT := 0;
	ST_ACTIVE_UNACK: DINT := 1;
	ST_ACTIVE_ACK: DINT := 2;
	ST_RTN_UNACK: DINT := 3;
	ST_LATCHED_UNACK: DINT := 4;
	ST_LATCHED_ACK: DINT := 5;
	ST_SHELVED: DINT := 6;
	ST_SUPPRESSED: DINT := 7;
	ST_OUT_OF_SERVICE: DINT := 8;
END_VAR

(*==========================================================================
Sets the Version of the Control Module on the HMI and in the Program.
==========================================================================
Date Last Updated: 10-1-2026
===========================================================================*)
//CFG_VERSION:= 1.0; // ORIGINAL
//CFG_VERSION := 2.0; //FIRST ALARM BLOCK (ARCHIVED AS archive/digital_alarm_v2.st)
//CFG_VERSION := 3.0; //ISA-18.2 STATE MODEL, SHELVING, OUT OF SERVICE, OFF-DELAY, CHATTER, DT TIME STAMPS
CFG_VERSION := 3.1; //RENAMED BG_ALM_DIG WITH IN_/CFG_/CMD_/STS_/VAL_/TS_ NAMES; NO LOGIC CHANGE

STS_ENABLED := IN_ENABLE;
IF NOT IN_ENABLE THEN
	JMP CLEAR_COMMANDS;
END_IF

IF CFG_USE_SRC_TIME THEN
	NOW := IN_SRC_TIME;
ELSE
	NOW := IN_CLOCK;
END_IF

(*===========================================================================
CONFIGURATION - Validate and map severity to priority
===========================================================================*)
VAL_DIAG := 0;
VAL_DIAG.2 := CFG_SEVERITY < 1 OR CFG_SEVERITY > 1000;
VAL_DIAG.3 := CFG_ON_DELAY_MS < 0 OR CFG_OFF_DELAY_MS < 0;
VAL_DIAG.4 := CFG_CHATTER_COUNT < 0 OR (CFG_CHATTER_COUNT > 0 AND CFG_CHATTER_WINDOW = T#0S);
STS_CFG_FAULT := VAL_DIAG.2 OR VAL_DIAG.3 OR VAL_DIAG.4;

IF CFG_SEVERITY <= 250 THEN
	VAL_PRIORITY := 4;
ELSIF CFG_SEVERITY <= 500 THEN
	VAL_PRIORITY := 3;
ELSIF CFG_SEVERITY <= 750 THEN
	VAL_PRIORITY := 2;
ELSE
	VAL_PRIORITY := 1;
END_IF

(*===========================================================================
CONDITION - Invert, hold on bad quality, then apply the on-delay and off-delay
===========================================================================*)
RAWCOND := IN_SIGNAL XOR CFG_INVERT;
STS_IN_FAULT := IN_FAULT;
IF IN_FAULT THEN
	RAWCOND := LASTGOODCOND;	// BAD DATA MUST NOT RAISE OR CLEAR THE ALARM
ELSE
	LASTGOODCOND := RAWCOND;
END_IF

ON_TMR(IN := RAWCOND AND NOT COND, PT := DINT_TO_TIME(MAX(CFG_ON_DELAY_MS, 0)));
OFF_TMR(IN := NOT RAWCOND AND COND, PT := DINT_TO_TIME(MAX(CFG_OFF_DELAY_MS, 0)));
IF ON_TMR.Q THEN
	COND := TRUE;
ELSIF OFF_TMR.Q THEN
	COND := FALSE;
END_IF
VAL_ON_DELAY_MS := TIME_TO_DINT(ON_TMR.ET);
STS_COND := COND;
COND_RISE(CLK := COND);
COND_FALL(CLK := COND);

(*===========================================================================
REQUESTS - Operator one-shots and logic rising edges
===========================================================================*)
PG_ACK_ONS(CLK := CMD_PG_ACK);
PG_RESET_ONS(CLK := CMD_PG_RESET);
PG_DISABLE_ONS(CLK := CMD_PG_DISABLE);
PG_ENABLE_ONS(CLK := CMD_PG_ENABLE);
PG_SUPPRESS_ONS(CLK := CMD_PG_SUPPRESS);
PG_UNSUPPRESS_ONS(CLK := CMD_PG_UNSUPPRESS);
PG_UNSHELVE_ONS(CLK := CMD_PG_UNSHELVE);

ACKCMD := CMD_OP_ACK OR PG_ACK_ONS.Q;
RESETCMD := CMD_OP_RESET OR PG_RESET_ONS.Q;
DISABLECMD := CMD_OP_DISABLE OR PG_DISABLE_ONS.Q;
ENABLECMD := CMD_OP_ENABLE OR PG_ENABLE_ONS.Q;
SUPPRESSCMD := CMD_OP_SUPPRESS OR PG_SUPPRESS_ONS.Q;
UNSUPPRESSCMD := CMD_OP_UNSUPPRESS OR PG_UNSUPPRESS_ONS.Q;
SHELVECMD := CMD_OP_SHELVE;
UNSHELVECMD := CMD_OP_UNSHELVE OR PG_UNSHELVE_ONS.Q;

(*===========================================================================
OUT OF SERVICE (ISA H) - Supersedes shelving
===========================================================================*)
IF DISABLECMD AND NOT STS_DISABLED THEN
	STS_DISABLED := TRUE;
	IF STS_SHELVED THEN
		STS_SHELVED := FALSE;
		TS_UNSHELVE := NOW;
	END_IF
END_IF
IF ENABLECMD THEN
	STS_DISABLED := FALSE;
END_IF

(*===========================================================================
SUPPRESSED BY DESIGN (ISA G)
===========================================================================*)
IF SUPPRESSCMD THEN
	STS_SUPPRESSED := TRUE;
END_IF
IF UNSUPPRESSCMD THEN
	STS_SUPPRESSED := FALSE;
END_IF

(*===========================================================================
SHELVING (ISA F) - Operator only, always time-limited by CFG_SHELVE_MAX.
A shelve request while shelved restarts the timer with the new duration.
===========================================================================*)
IF SHELVECMD THEN
	IF STS_DISABLED OR CFG_SHELVE_MAX = T#0S OR (CMD_SHELVE_ONESHOT AND NOT COND) THEN
		SHELVEREJECTED := TRUE;
	ELSE
		IF CMD_SHELVE_TIME = T#0S OR CMD_SHELVE_TIME > CFG_SHELVE_MAX THEN
			SHELVEPT := CFG_SHELVE_MAX;
		ELSE
			SHELVEPT := CMD_SHELVE_TIME;
		END_IF
		STS_SHELVED := TRUE;
		SHELVEDONESHOT := CMD_SHELVE_ONESHOT;
		SHELVEREJECTED := FALSE;
		TS_SHELVE := NOW;
		TS_SHELVE_EXPIRY := ADD_DT_TIME(NOW, SHELVEPT);
		SHELVE_TMR(IN := FALSE);
	END_IF
END_IF

SHELVE_TMR(IN := STS_SHELVED, PT := SHELVEPT);
IF STS_SHELVED AND (UNSHELVECMD OR SHELVE_TMR.Q OR (SHELVEDONESHOT AND COND_FALL.Q)) THEN
	STS_SHELVED := FALSE;
	TS_UNSHELVE := NOW;
	SHELVE_TMR(IN := FALSE);
END_IF

IF STS_SHELVED THEN
	VAL_SHELVE_LEFT := SHELVEPT - SHELVE_TMR.ET;
ELSE
	VAL_SHELVE_LEFT := T#0S;
END_IF

(*===========================================================================
ALARM STATE MACHINE (ISA A-E)
While shelved, suppressed or out of service the alarm is held at NORMAL, so an
active condition re-annunciates as ACTIVE_UNACK when the alarm is returned.
===========================================================================*)
IF STS_DISABLED OR STS_SUPPRESSED OR STS_SHELVED THEN
	ALMSTATE := ST_NORMAL;
ELSE
	// CONDITION CHANGES
	CASE ALMSTATE OF
	ST_NORMAL, ST_RTN_UNACK, ST_LATCHED_UNACK, ST_LATCHED_ACK:
		IF COND THEN
			ALMSTATE := ST_ACTIVE_UNACK;
			VAL_COUNT := VAL_COUNT + 1;
			TS_ALM := NOW;
		END_IF
	ST_ACTIVE_UNACK:
		IF NOT COND THEN
			TS_RTN := NOW;
			IF CFG_LATCH THEN
				ALMSTATE := ST_LATCHED_UNACK;
			ELSE
				ALMSTATE := ST_RTN_UNACK;
			END_IF
		END_IF
	ST_ACTIVE_ACK:
		IF NOT COND THEN
			TS_RTN := NOW;
			IF CFG_LATCH THEN
				ALMSTATE := ST_LATCHED_ACK;
			ELSE
				ALMSTATE := ST_NORMAL;
			END_IF
		END_IF
	END_CASE

	// ACKNOWLEDGE - IMPLICIT WHEN NO ACKNOWLEDGEMENT IS REQUIRED
	IF ACKCMD OR NOT CFG_ACK_REQ THEN
		CASE ALMSTATE OF
		ST_ACTIVE_UNACK:
			ALMSTATE := ST_ACTIVE_ACK;
			TS_ACK := NOW;
		ST_RTN_UNACK:
			ALMSTATE := ST_NORMAL;
			TS_ACK := NOW;
		ST_LATCHED_UNACK:
			ALMSTATE := ST_LATCHED_ACK;
			TS_ACK := NOW;
		END_CASE
	END_IF

	// RESET - ONLY A LATCHED ALARM THAT IS BACK TO NORMAL AND ACKNOWLEDGED.
	// AN ACK AND RESET IN THE SAME SCAN CLEARS A LATCHED_UNACK ALARM.
	IF RESETCMD AND ALMSTATE = ST_LATCHED_ACK THEN
		ALMSTATE := ST_NORMAL;
		TS_RESET := NOW;
	END_IF
END_IF

(*===========================================================================
CHATTER - CFG_CHATTER_COUNT or more activations within one CFG_CHATTER_WINDOW.
Cleared at the end of a window with fewer activations.
===========================================================================*)
IF CFG_CHATTER_COUNT > 0 THEN
	CHATTER_TMR(IN := NOT CHATTER_TMR.Q, PT := CFG_CHATTER_WINDOW);
	IF COND_RISE.Q THEN
		CHATTERACC := CHATTERACC + 1;
	END_IF
	IF CHATTERACC >= CFG_CHATTER_COUNT THEN
		STS_CHATTER := TRUE;
	END_IF
	IF CHATTER_TMR.Q THEN
		STS_CHATTER := CHATTERACC >= CFG_CHATTER_COUNT;
		CHATTERACC := 0;
	END_IF
ELSE
	CHATTER_TMR(IN := FALSE);
	CHATTERACC := 0;
	STS_CHATTER := FALSE;
END_IF

(*===========================================================================
ALARM COUNT
===========================================================================*)
COUNTRESET_ONS(CLK := CMD_COUNT_RESET);
IF COUNTRESET_ONS.Q THEN
	VAL_COUNT := 0;
	TS_COUNT_RESET := NOW;
END_IF

(*===========================================================================
OUTPUT UPDATES
===========================================================================*)
STS_ALM := ALMSTATE = ST_ACTIVE_UNACK OR ALMSTATE = ST_ACTIVE_ACK
	OR ALMSTATE = ST_LATCHED_UNACK OR ALMSTATE = ST_LATCHED_ACK;
STS_UNACKED := ALMSTATE = ST_ACTIVE_UNACK OR ALMSTATE = ST_RTN_UNACK OR ALMSTATE = ST_LATCHED_UNACK;
STS_ACKED := NOT STS_UNACKED;
STS_ALM_UNACK := STS_ALM AND STS_UNACKED;

IF STS_DISABLED THEN
	VAL_STATE := ST_OUT_OF_SERVICE;
ELSIF STS_SUPPRESSED THEN
	VAL_STATE := ST_SUPPRESSED;
ELSIF STS_SHELVED THEN
	VAL_STATE := ST_SHELVED;
ELSE
	VAL_STATE := ALMSTATE;
END_IF

VAL_DIAG.0 := STS_CFG_FAULT;
VAL_DIAG.1 := IN_FAULT;
VAL_DIAG.5 := SHELVEREJECTED;
VAL_DIAG.6 := STS_CHATTER;

(*===========================================================================
CLEAR OPERATOR REQUESTS - They are one-shot
===========================================================================*)
CLEAR_COMMANDS:
CMD_OP_ACK := FALSE;
CMD_OP_RESET := FALSE;
CMD_OP_DISABLE := FALSE;
CMD_OP_ENABLE := FALSE;
CMD_OP_SUPPRESS := FALSE;
CMD_OP_UNSUPPRESS := FALSE;
CMD_OP_SHELVE := FALSE;
CMD_OP_UNSHELVE := FALSE;

END_FUNCTION_BLOCK
